// TIA Portal project "Elevator" (V15)

(* hardware
DEVICE "S7-1200 station_1"  S7-1200 Station
   slot 0: "Rack_0"  S7-1200 Rack  Rack  V1.0
   slot 1: "PLC_1"  CPU 1215C DC/DC/Rly  6ES7 215-1HG40-0XB0  V4.2
DEVICE "HMI_1"  KTP700 Basic PN
   slot 0: "HMI_1"  KTP700 Basic PN  6AV2 123-2GB03-0AX0  15.0.0.0
   slot 1: "HMI_RT_1"  KTP700 Basic PN  6AV2 123-2GB03-0AX0  15.0.0.0
   slot 5: "HMI_1.IE_CP_1"  PROFINET Interface  15.0.0.0
      slot 1: "PROFINET Interface_1"  PROFINET Interface
         slot 1: "Port_1"  Port
*)

// ===== PLC "PLC_1"  CPU 1215C DC/DC/Rly =====

VAR_GLOBAL   // PLC tag table "Default tag table"
   "asansor_tus_F1" AT %I4.0 : Bool;
   "kat_cagri_F1" AT %I4.5 : Bool;
   "kat_1" AT %M0.0 : Bool;
   "asansor_tus_F2" AT %I4.1 : Bool;
   "kat_cagri_F2" AT %I4.6 : Bool;
   "kat_2" AT %M0.1 : Bool;
   "asansor_tus_F3" AT %I4.2 : Bool;
   "kat_cagri_F3" AT %I4.7 : Bool;
   "kat_3" AT %M0.2 : Bool;
   "asansor_tus_F4" AT %I4.3 : Bool;
   "kat_cagri_F4" AT %I5.0 : Bool;
   "kat_4" AT %M0.3 : Bool;
   "Clock_1Hz" AT %M100.5 : Bool;
   "Motor_Yukari" AT %Q7.1 : Bool;
   "Motor_Asagi" AT %Q7.2 : Bool;
   "bas_sayaci" AT %MW10 : UInt;
   "System_Byte" AT %MB100 : Byte;
   "FirstScan" AT %M100.0 : Bool;
   "DiagStatusUpdate" AT %M100.1 : Bool;
   "AlwaysTRUE" AT %M100.2 : Bool;
   "AlwaysFALSE" AT %M100.3 : Bool;
   "Clock_Byte" AT %MB100 : Byte;
   "Clock_10Hz" AT %M100.0 : Bool;
   "Clock_5Hz" AT %M100.1 : Bool;
   "Clock_2.5Hz" AT %M100.2 : Bool;
   "Clock_2Hz" AT %M100.3 : Bool;
   "Clock_1.25Hz" AT %M100.4 : Bool;
   "Clock_0.625Hz" AT %M100.6 : Bool;
   "Clock_0.5Hz" AT %M100.7 : Bool;
   "F1_sensor" AT %I6.0 : Bool;
   "F2_sensor" AT %I6.1 : Bool;
   "F4_sensor" AT %I6.3 : Bool;
   "F3_sensor" AT %I6.2 : Bool;
   "F5_sensor" AT %I6.4 : Bool;
   "yon_yukari" AT %M0.5 : Bool;
   "yon_asagi" AT %M0.6 : Bool;
   "kat_5" AT %M0.4 : Bool;
   "asansor_tus_F5" AT %I4.4 : Bool;
   "kat_cagri_F5" AT %I5.1 : Bool;
   "kapi_kapaniyor" AT %M2.1 : Bool;
   "kapi_motoru" AT %Q7.0 : Bool;
   "kapi_acik_F3" AT %M1.2 : Bool;
   "kapi_kapandi" AT %M2.0 : Bool;
   "kapi_acik_F4" AT %M1.3 : Bool;
   "kapi_acik_F2" AT %M1.1 : Bool;
   "kapi_acik_F1" AT %M1.0 : Bool;
   "kapi_acik_F5" AT %M1.4 : Bool;
   "acma_tusu" AT %I5.2 : Bool;
   "engel_sensor" AT %I5.4 : Bool;
   "agirlik_sensor" AT %I5.5 : Bool;
   "kapi_tekrar_acildi" AT %M2.3 : Bool;
   "kapama_tusu" AT %I5.3 : Bool;
   "Tag_1" AT %M1.5 : Bool;
   "Tag_2" AT %M1.6 : Bool;
END_VAR

// folder: System blocks/Program resources

DATA_BLOCK "delay_reset5"   // DB1
{ S7_Optimized_Access := 'TRUE' }
AUTHOR : Simatic
FAMILY : IEC
NAME : IEC_TMR
VERSION : 1.0
// stored: InstanceOfName IEC_TIMER
"IEC_TIMER"
BEGIN
END_DATA_BLOCK

DATA_BLOCK "delay_reset4"   // DB2
{ S7_Optimized_Access := 'TRUE' }
AUTHOR : Simatic
FAMILY : IEC
NAME : IEC_TMR
VERSION : 1.0
// stored: InstanceOfName IEC_TIMER
"IEC_TIMER"
BEGIN
END_DATA_BLOCK

DATA_BLOCK "delay_reset3"   // DB3
{ S7_Optimized_Access := 'TRUE' }
AUTHOR : Simatic
FAMILY : IEC
NAME : IEC_TMR
VERSION : 1.0
// stored: InstanceOfName IEC_TIMER
"IEC_TIMER"
BEGIN
END_DATA_BLOCK

DATA_BLOCK "delay_reset2"   // DB4
{ S7_Optimized_Access := 'TRUE' }
AUTHOR : Simatic
FAMILY : IEC
NAME : IEC_TMR
VERSION : 1.0
// stored: InstanceOfName IEC_TIMER
"IEC_TIMER"
BEGIN
END_DATA_BLOCK

DATA_BLOCK "kapi_acik_zamani"   // DB5
{ S7_Optimized_Access := 'TRUE' }
AUTHOR : Simatic
FAMILY : IEC
NAME : IEC_TMR
VERSION : 1.0
// stored: InstanceOfName IEC_TIMER
"IEC_TIMER"
BEGIN
END_DATA_BLOCK

DATA_BLOCK "kapi_kapanma_zamani"   // DB6
{ S7_Optimized_Access := 'TRUE' }
AUTHOR : Simatic
FAMILY : IEC
NAME : IEC_TMR
VERSION : 1.0
// stored: InstanceOfName IEC_TIMER
"IEC_TIMER"
BEGIN
END_DATA_BLOCK

DATA_BLOCK "reset_acilma_zamani"   // DB7
{ S7_Optimized_Access := 'TRUE' }
AUTHOR : Simatic
FAMILY : IEC
NAME : IEC_TMR
VERSION : 1.0
// stored: InstanceOfName IEC_TIMER
"IEC_TIMER"
BEGIN
END_DATA_BLOCK

DATA_BLOCK "reset_kapama_tusu"   // DB8
{ S7_Optimized_Access := 'TRUE' }
AUTHOR : Simatic
FAMILY : IEC
NAME : IEC_TMR
VERSION : 1.0
// stored: InstanceOfName IEC_TIMER
"IEC_TIMER"
BEGIN
END_DATA_BLOCK

DATA_BLOCK "delay_reset1"   // DB9
{ S7_Optimized_Access := 'TRUE' }
AUTHOR : Simatic
FAMILY : IEC
NAME : IEC_TMR
VERSION : 1.0
// stored: InstanceOfName IEC_TIMER
"IEC_TIMER"
BEGIN
END_DATA_BLOCK

// folder: (top level)

ORGANIZATION_BLOCK "Main"   // OB1, LAD, ProgramCycle
TITLE = "Main Program Sweep (Cycle)"
{ S7_Optimized_Access := 'TRUE' }
VERSION : 0.1
   VAR_INPUT
      Initial_Call : Bool;   // Initial call of this OB
      Remanence : Bool;   // =True, if remanent data are available
   END_VAR
   VAR_TEMP   // added for the SCL form of the ladder/FBD networks
      _w1 : Bool;
      _w2 : Bool;
      _w3 : Bool;
      _w4 : Bool;
      _w5 : Bool;
   END_VAR
BEGIN

REGION Network 1: Asansör Çağrıları
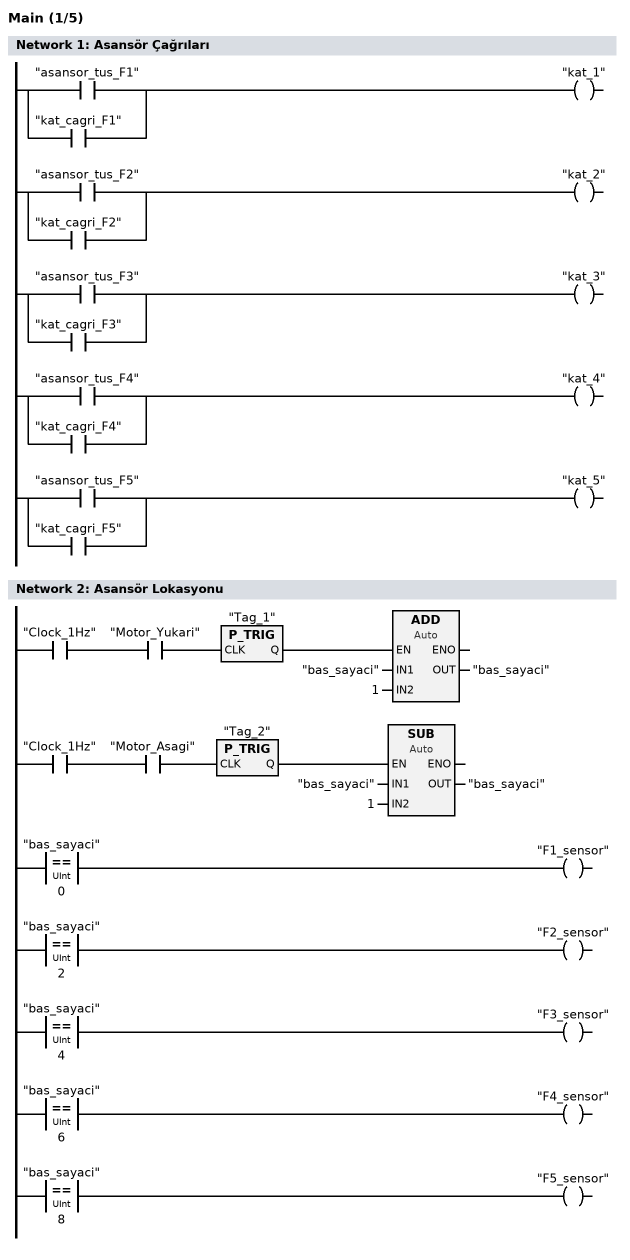
   RUNG wire#powerrail
      Contact( "asansor_tus_F1" )
      wire#w1
      Coil( "kat_1" )
   END_RUNG
   RUNG wire#powerrail
      Contact( "kat_cagri_F1" )
   END_RUNG wire#w1
   RUNG wire#powerrail
      Contact( "asansor_tus_F2" )
      wire#w2
      Coil( "kat_2" )
   END_RUNG
   RUNG wire#powerrail
      Contact( "kat_cagri_F2" )
   END_RUNG wire#w2
   RUNG wire#powerrail
      Contact( "asansor_tus_F3" )
      wire#w3
      Coil( "kat_3" )
   END_RUNG
   RUNG wire#powerrail
      Contact( "kat_cagri_F3" )
   END_RUNG wire#w3
   RUNG wire#powerrail
      Contact( "asansor_tus_F4" )
      wire#w4
      Coil( "kat_4" )
   END_RUNG
   RUNG wire#powerrail
      Contact( "kat_cagri_F4" )
   END_RUNG wire#w4
   RUNG wire#powerrail
      Contact( "asansor_tus_F5" )
      wire#w5
      Coil( "kat_5" )
   END_RUNG
   RUNG wire#powerrail
      Contact( "kat_cagri_F5" )
   END_RUNG wire#w5
   // the same network as SCL:
   "kat_1" := "asansor_tus_F1" OR "kat_cagri_F1";
   "kat_2" := "asansor_tus_F2" OR "kat_cagri_F2";
   "kat_3" := "asansor_tus_F3" OR "kat_cagri_F3";
   "kat_4" := "asansor_tus_F4" OR "kat_cagri_F4";
   "kat_5" := "asansor_tus_F5" OR "kat_cagri_F5";
END_REGION

REGION Network 2: Asansör Lokasyonu
   RUNG wire#powerrail
      Contact( "Clock_1Hz" )
      Contact( "Motor_Yukari" )
      P_Trig( "Tag_1" )
      Add(in1 := "bas_sayaci", in2 := 1, out => "bas_sayaci")
   END_RUNG
   RUNG wire#powerrail
      Contact( "Clock_1Hz" )
      Contact( "Motor_Asagi" )
      P_Trig( "Tag_2" )
      Sub(in1 := "bas_sayaci", in2 := 1, out => "bas_sayaci")
   END_RUNG
   RUNG wire#powerrail
      { S7_Templates := "SrcType := UInt" } EQ_Contact(in1 := "bas_sayaci", in2 := 0)
      Coil( "F1_sensor" )
   END_RUNG
   RUNG wire#powerrail
      { S7_Templates := "SrcType := UInt" } EQ_Contact(in1 := "bas_sayaci", in2 := 2)
      Coil( "F2_sensor" )
   END_RUNG
   RUNG wire#powerrail
      { S7_Templates := "SrcType := UInt" } EQ_Contact(in1 := "bas_sayaci", in2 := 4)
      Coil( "F3_sensor" )
   END_RUNG
   RUNG wire#powerrail
      { S7_Templates := "SrcType := UInt" } EQ_Contact(in1 := "bas_sayaci", in2 := 6)
      Coil( "F4_sensor" )
   END_RUNG
   RUNG wire#powerrail
      { S7_Templates := "SrcType := UInt" } EQ_Contact(in1 := "bas_sayaci", in2 := 8)
      Coil( "F5_sensor" )
   END_RUNG
   // the same network as SCL:
   #_w1 := "Clock_1Hz" AND "Motor_Yukari";
   #_w2 := #_w1 AND NOT "Tag_1";   // rising edge
   "Tag_1" := #_w1;
   IF #_w2 THEN "bas_sayaci" := "bas_sayaci" + 1; END_IF;
   #_w3 := "Clock_1Hz" AND "Motor_Asagi";
   #_w4 := #_w3 AND NOT "Tag_2";   // rising edge
   "Tag_2" := #_w3;
   IF #_w4 THEN "bas_sayaci" := "bas_sayaci" - 1; END_IF;
   "F1_sensor" := "bas_sayaci" = 0;
   "F2_sensor" := "bas_sayaci" = 2;
   "F3_sensor" := "bas_sayaci" = 4;
   "F4_sensor" := "bas_sayaci" = 6;
   "F5_sensor" := "bas_sayaci" = 8;
END_REGION

REGION Network 3: Asansör Yönelimi
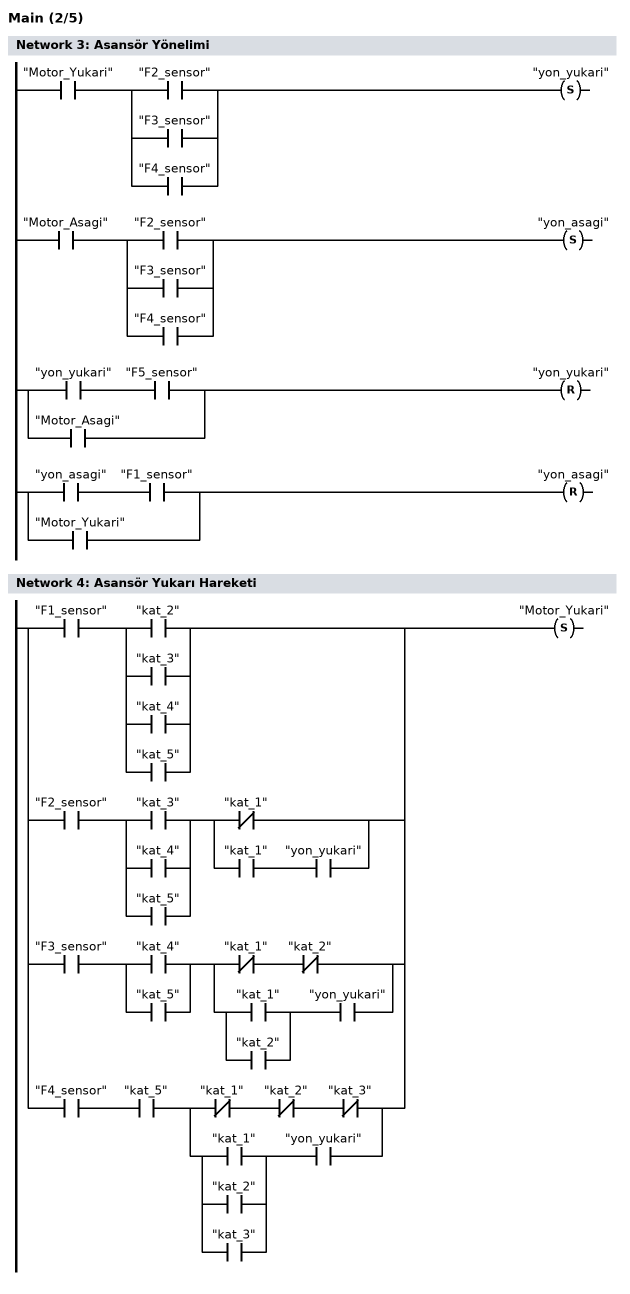
   RUNG wire#powerrail
      Contact( "Motor_Yukari" )
      wire#w1
      Contact( "F2_sensor" )
      wire#w2
      S_Coil( "yon_yukari" )
   END_RUNG
   RUNG wire#w1
      Contact( "F3_sensor" )
   END_RUNG wire#w2
   RUNG wire#w1
      Contact( "F4_sensor" )
   END_RUNG wire#w2
   RUNG wire#powerrail
      Contact( "Motor_Asagi" )
      wire#w3
      Contact( "F2_sensor" )
      wire#w4
      S_Coil( "yon_asagi" )
   END_RUNG
   RUNG wire#w3
      Contact( "F3_sensor" )
   END_RUNG wire#w4
   RUNG wire#w3
      Contact( "F4_sensor" )
   END_RUNG wire#w4
   RUNG wire#powerrail
      Contact( "yon_yukari" )
      Contact( "F5_sensor" )
      wire#w5
      R_Coil( "yon_yukari" )
   END_RUNG
   RUNG wire#powerrail
      Contact( "Motor_Asagi" )
   END_RUNG wire#w5
   RUNG wire#powerrail
      Contact( "yon_asagi" )
      Contact( "F1_sensor" )
      wire#w6
      R_Coil( "yon_asagi" )
   END_RUNG
   RUNG wire#powerrail
      Contact( "Motor_Yukari" )
   END_RUNG wire#w6
   // the same network as SCL:
   IF "Motor_Yukari" AND ("F2_sensor" OR "F3_sensor" OR "F4_sensor") THEN "yon_yukari" := TRUE; END_IF;
   IF "Motor_Asagi" AND ("F2_sensor" OR "F3_sensor" OR "F4_sensor") THEN "yon_asagi" := TRUE; END_IF;
   IF ("yon_yukari" AND "F5_sensor") OR "Motor_Asagi" THEN "yon_yukari" := FALSE; END_IF;
   IF ("yon_asagi" AND "F1_sensor") OR "Motor_Yukari" THEN "yon_asagi" := FALSE; END_IF;
END_REGION

REGION Network 4: Asansör Yukarı Hareketi
   RUNG wire#powerrail
      Contact( "F1_sensor" )
      wire#w1
      Contact( "kat_2" )
      wire#w2
      S_Coil( "Motor_Yukari" )
   END_RUNG
   RUNG wire#w1
      Contact( "kat_3" )
   END_RUNG wire#w2
   RUNG wire#w1
      Contact( "kat_4" )
   END_RUNG wire#w2
   RUNG wire#w1
      Contact( "kat_5" )
   END_RUNG wire#w2
   RUNG wire#powerrail
      Contact( "F2_sensor" )
      wire#w3
      Contact( "kat_3" )
      wire#w4
      I_Contact( "kat_1" )
   END_RUNG wire#w2
   RUNG wire#w3
      Contact( "kat_4" )
   END_RUNG wire#w4
   RUNG wire#w3
      Contact( "kat_5" )
   END_RUNG wire#w4
   RUNG wire#w4
      Contact( "kat_1" )
      Contact( "yon_yukari" )
   END_RUNG wire#w2
   RUNG wire#powerrail
      Contact( "F3_sensor" )
      wire#w5
      Contact( "kat_4" )
      wire#w6
      I_Contact( "kat_1" )
      I_Contact( "kat_2" )
   END_RUNG wire#w2
   RUNG wire#w5
      Contact( "kat_5" )
   END_RUNG wire#w6
   RUNG wire#w6
      Contact( "kat_1" )
      wire#w7
      Contact( "yon_yukari" )
   END_RUNG wire#w2
   RUNG wire#w6
      Contact( "kat_2" )
   END_RUNG wire#w7
   RUNG wire#powerrail
      Contact( "F4_sensor" )
      Contact( "kat_5" )
      wire#w8
      I_Contact( "kat_1" )
      I_Contact( "kat_2" )
      I_Contact( "kat_3" )
   END_RUNG wire#w2
   RUNG wire#w8
      Contact( "kat_1" )
      wire#w9
      Contact( "yon_yukari" )
   END_RUNG wire#w2
   RUNG wire#w8
      Contact( "kat_2" )
   END_RUNG wire#w9
   RUNG wire#w8
      Contact( "kat_3" )
   END_RUNG wire#w9
   // the same network as SCL:
   IF ("F1_sensor" AND ("kat_2" OR "kat_3" OR "kat_4" OR "kat_5")) OR ("F2_sensor" AND ("kat_3" OR "kat_4" OR "kat_5") AND (NOT "kat_1" OR ("kat_1" AND "yon_yukari"))) OR ("F3_sensor" AND ("kat_4" OR "kat_5") AND ((NOT "kat_1" AND NOT "kat_2") OR (("kat_1" OR "kat_2") AND "yon_yukari"))) OR ("F4_sensor" AND "kat_5" AND ((NOT "kat_1" AND NOT "kat_2" AND NOT "kat_3") OR (("kat_1" OR "kat_2" OR "kat_3") AND "yon_yukari"))) THEN
       "Motor_Yukari" := TRUE;
   END_IF;
END_REGION

REGION Network 5: Asansör Aşağı Hareketi
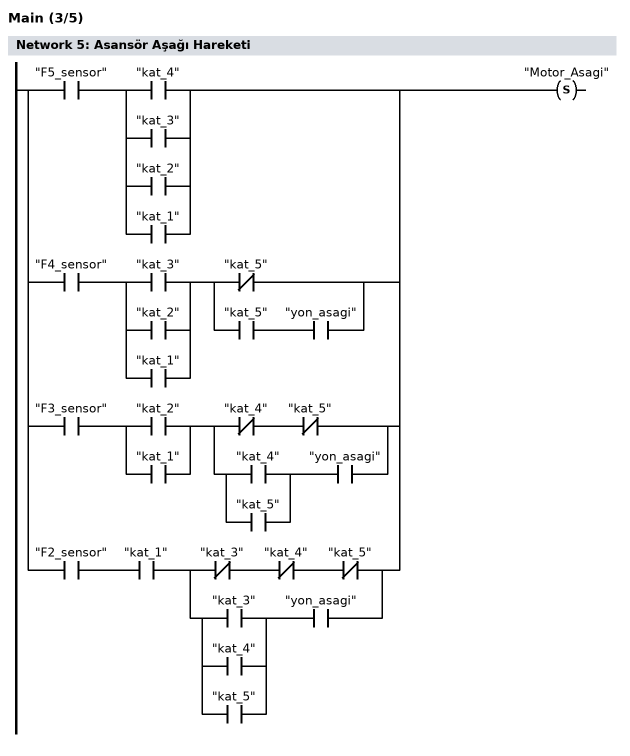
   RUNG wire#powerrail
      Contact( "F5_sensor" )
      wire#w1
      Contact( "kat_4" )
      wire#w2
      S_Coil( "Motor_Asagi" )
   END_RUNG
   RUNG wire#w1
      Contact( "kat_3" )
   END_RUNG wire#w2
   RUNG wire#w1
      Contact( "kat_2" )
   END_RUNG wire#w2
   RUNG wire#w1
      Contact( "kat_1" )
   END_RUNG wire#w2
   RUNG wire#powerrail
      Contact( "F4_sensor" )
      wire#w3
      Contact( "kat_3" )
      wire#w4
      I_Contact( "kat_5" )
   END_RUNG wire#w2
   RUNG wire#w3
      Contact( "kat_2" )
   END_RUNG wire#w4
   RUNG wire#w3
      Contact( "kat_1" )
   END_RUNG wire#w4
   RUNG wire#w4
      Contact( "kat_5" )
      Contact( "yon_asagi" )
   END_RUNG wire#w2
   RUNG wire#powerrail
      Contact( "F3_sensor" )
      wire#w5
      Contact( "kat_2" )
      wire#w6
      I_Contact( "kat_4" )
      I_Contact( "kat_5" )
   END_RUNG wire#w2
   RUNG wire#w5
      Contact( "kat_1" )
   END_RUNG wire#w6
   RUNG wire#w6
      Contact( "kat_4" )
      wire#w7
      Contact( "yon_asagi" )
   END_RUNG wire#w2
   RUNG wire#w6
      Contact( "kat_5" )
   END_RUNG wire#w7
   RUNG wire#powerrail
      Contact( "F2_sensor" )
      Contact( "kat_1" )
      wire#w8
      I_Contact( "kat_3" )
      I_Contact( "kat_4" )
      I_Contact( "kat_5" )
   END_RUNG wire#w2
   RUNG wire#w8
      Contact( "kat_3" )
      wire#w9
      Contact( "yon_asagi" )
   END_RUNG wire#w2
   RUNG wire#w8
      Contact( "kat_4" )
   END_RUNG wire#w9
   RUNG wire#w8
      Contact( "kat_5" )
   END_RUNG wire#w9
   // the same network as SCL:
   IF ("F5_sensor" AND ("kat_4" OR "kat_3" OR "kat_2" OR "kat_1")) OR ("F4_sensor" AND ("kat_3" OR "kat_2" OR "kat_1") AND (NOT "kat_5" OR ("kat_5" AND "yon_asagi"))) OR ("F3_sensor" AND ("kat_2" OR "kat_1") AND ((NOT "kat_4" AND NOT "kat_5") OR (("kat_4" OR "kat_5") AND "yon_asagi"))) OR ("F2_sensor" AND "kat_1" AND ((NOT "kat_3" AND NOT "kat_4" AND NOT "kat_5") OR (("kat_3" OR "kat_4" OR "kat_5") AND "yon_asagi"))) THEN
       "Motor_Asagi" := TRUE;
   END_IF;
END_REGION

REGION Network 6: Asansör Durma - Kapı Açılması
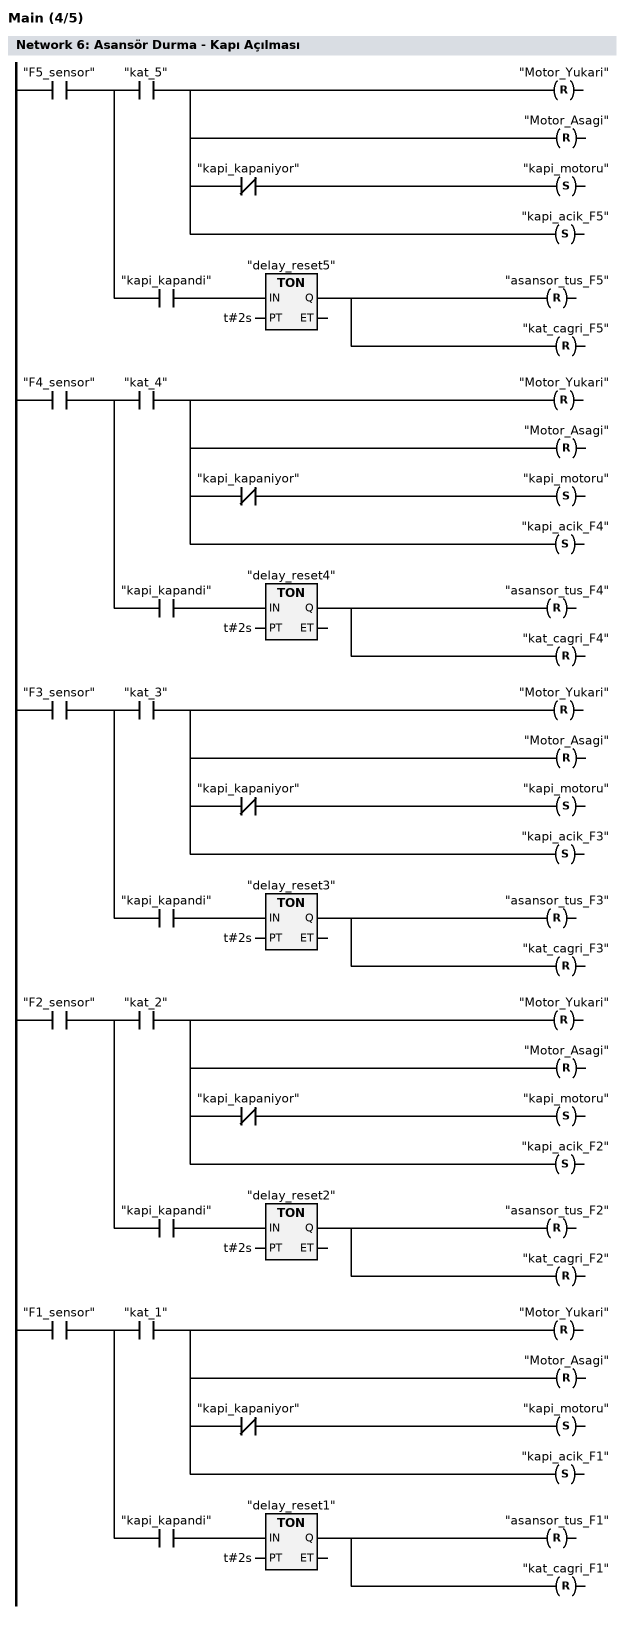
   #_w1 := "F5_sensor" AND "kat_5";
   IF #_w1 THEN
       "Motor_Yukari" := FALSE;
       "Motor_Asagi" := FALSE;
   END_IF;
   IF #_w1 AND NOT "kapi_kapaniyor" THEN "kapi_motoru" := TRUE; END_IF;
   IF #_w1 THEN "kapi_acik_F5" := TRUE; END_IF;
   "delay_reset5".TON(IN := "F5_sensor" AND "kapi_kapandi", PT := t#2s);
   IF "delay_reset5".Q THEN
       "asansor_tus_F5" := FALSE;
       "kat_cagri_F5" := FALSE;
   END_IF;
   #_w2 := "F4_sensor" AND "kat_4";
   IF #_w2 THEN
       "Motor_Yukari" := FALSE;
       "Motor_Asagi" := FALSE;
   END_IF;
   IF #_w2 AND NOT "kapi_kapaniyor" THEN "kapi_motoru" := TRUE; END_IF;
   IF #_w2 THEN "kapi_acik_F4" := TRUE; END_IF;
   "delay_reset4".TON(IN := "F4_sensor" AND "kapi_kapandi", PT := t#2s);
   IF "delay_reset4".Q THEN
       "asansor_tus_F4" := FALSE;
       "kat_cagri_F4" := FALSE;
   END_IF;
   #_w3 := "F3_sensor" AND "kat_3";
   IF #_w3 THEN
       "Motor_Yukari" := FALSE;
       "Motor_Asagi" := FALSE;
   END_IF;
   IF #_w3 AND NOT "kapi_kapaniyor" THEN "kapi_motoru" := TRUE; END_IF;
   IF #_w3 THEN "kapi_acik_F3" := TRUE; END_IF;
   "delay_reset3".TON(IN := "F3_sensor" AND "kapi_kapandi", PT := t#2s);
   IF "delay_reset3".Q THEN
       "asansor_tus_F3" := FALSE;
       "kat_cagri_F3" := FALSE;
   END_IF;
   #_w4 := "F2_sensor" AND "kat_2";
   IF #_w4 THEN
       "Motor_Yukari" := FALSE;
       "Motor_Asagi" := FALSE;
   END_IF;
   IF #_w4 AND NOT "kapi_kapaniyor" THEN "kapi_motoru" := TRUE; END_IF;
   IF #_w4 THEN "kapi_acik_F2" := TRUE; END_IF;
   "delay_reset2".TON(IN := "F2_sensor" AND "kapi_kapandi", PT := t#2s);
   IF "delay_reset2".Q THEN
       "asansor_tus_F2" := FALSE;
       "kat_cagri_F2" := FALSE;
   END_IF;
   #_w5 := "F1_sensor" AND "kat_1";
   IF #_w5 THEN
       "Motor_Yukari" := FALSE;
       "Motor_Asagi" := FALSE;
   END_IF;
   IF #_w5 AND NOT "kapi_kapaniyor" THEN "kapi_motoru" := TRUE; END_IF;
   IF #_w5 THEN "kapi_acik_F1" := TRUE; END_IF;
   "delay_reset1".TON(IN := "F1_sensor" AND "kapi_kapandi", PT := t#2s);
   IF "delay_reset1".Q THEN
       "asansor_tus_F1" := FALSE;
       "kat_cagri_F1" := FALSE;
   END_IF;
END_REGION

REGION Network 7: Asansör Kapı Kapanması
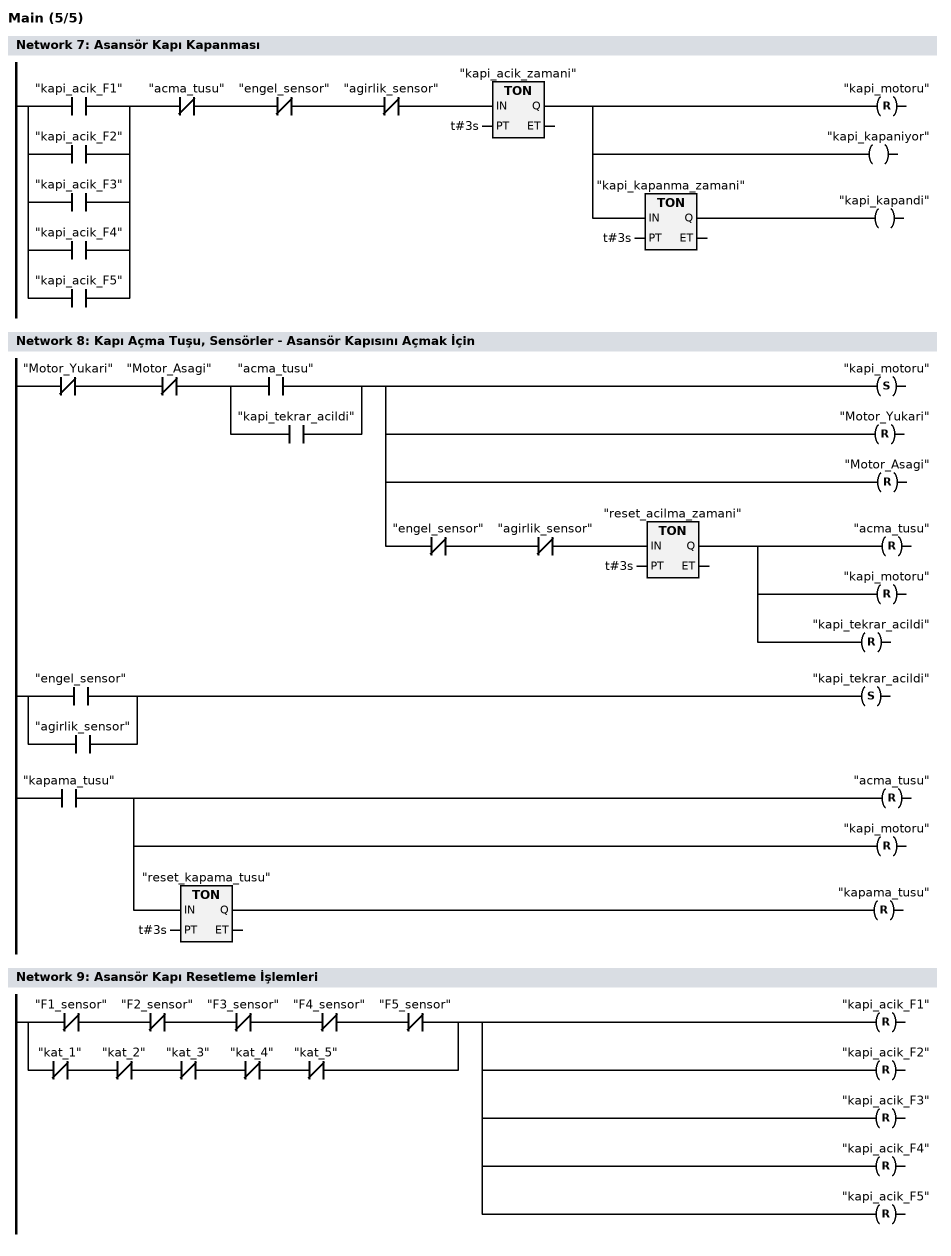
   "kapi_acik_zamani".TON(IN := ("kapi_acik_F1" OR "kapi_acik_F2" OR "kapi_acik_F3" OR "kapi_acik_F4" OR "kapi_acik_F5") AND NOT "acma_tusu" AND NOT "engel_sensor" AND NOT "agirlik_sensor",
                          PT := t#3s);
   IF "kapi_acik_zamani".Q THEN "kapi_motoru" := FALSE; END_IF;
   "kapi_kapaniyor" := "kapi_acik_zamani".Q;
   "kapi_kapanma_zamani".TON(IN := "kapi_acik_zamani".Q, PT := t#3s);
   "kapi_kapandi" := "kapi_kapanma_zamani".Q;
END_REGION

REGION Network 8: Kapı Açma Tuşu, Sensörler - Asansör Kapısını Açmak İçin
   #_w1 := NOT "Motor_Yukari" AND NOT "Motor_Asagi" AND ("acma_tusu" OR "kapi_tekrar_acildi");
   IF #_w1 THEN
       "kapi_motoru" := TRUE;
       "Motor_Yukari" := FALSE;
       "Motor_Asagi" := FALSE;
   END_IF;
   "reset_acilma_zamani".TON(IN := #_w1 AND NOT "engel_sensor" AND NOT "agirlik_sensor", PT := t#3s);
   IF "reset_acilma_zamani".Q THEN
       "acma_tusu" := FALSE;
       "kapi_motoru" := FALSE;
       "kapi_tekrar_acildi" := FALSE;
   END_IF;
   IF "engel_sensor" OR "agirlik_sensor" THEN "kapi_tekrar_acildi" := TRUE; END_IF;
   IF "kapama_tusu" THEN
       "acma_tusu" := FALSE;
       "kapi_motoru" := FALSE;
   END_IF;
   "reset_kapama_tusu".TON(IN := "kapama_tusu", PT := t#3s);
   IF "reset_kapama_tusu".Q THEN "kapama_tusu" := FALSE; END_IF;
END_REGION

REGION Network 9: Asansör Kapı Resetleme İşlemleri
   RUNG wire#powerrail
      I_Contact( "F1_sensor" )
      I_Contact( "F2_sensor" )
      I_Contact( "F3_sensor" )
      I_Contact( "F4_sensor" )
      I_Contact( "F5_sensor" )
      wire#w1
      R_Coil( "kapi_acik_F1" )
   END_RUNG
   RUNG wire#powerrail
      I_Contact( "kat_1" )
      I_Contact( "kat_2" )
      I_Contact( "kat_3" )
      I_Contact( "kat_4" )
      I_Contact( "kat_5" )
   END_RUNG wire#w1
   RUNG wire#w1
      R_Coil( "kapi_acik_F2" )
   END_RUNG
   RUNG wire#w1
      R_Coil( "kapi_acik_F3" )
   END_RUNG
   RUNG wire#w1
      R_Coil( "kapi_acik_F4" )
   END_RUNG
   RUNG wire#w1
      R_Coil( "kapi_acik_F5" )
   END_RUNG
   // the same network as SCL:
   IF (NOT "F1_sensor" AND NOT "F2_sensor" AND NOT "F3_sensor" AND NOT "F4_sensor" AND NOT "F5_sensor") OR (NOT "kat_1" AND NOT "kat_2" AND NOT "kat_3" AND NOT "kat_4" AND NOT "kat_5") THEN
       "kapi_acik_F1" := FALSE;
       "kapi_acik_F2" := FALSE;
       "kapi_acik_F3" := FALSE;
       "kapi_acik_F4" := FALSE;
       "kapi_acik_F5" := FALSE;
   END_IF;
END_REGION
END_ORGANIZATION_BLOCK

(* ===== HMI "HMI_RT_1" =====
system functions are stored by id; their names below are inferred from use
connection "HMI_Connection_1": ETHERNET, SMART_S7_1200_OMS

HMI tags "Default tag table"
   "Tag_ScreenNumber" : UInt, internal
   "kat_1" : Bool = PLC kat_1 AT %M0.0, 1 s
   "kat_2" : Bool = PLC kat_2 AT %M0.1, 1 s
   "kat_3" : Bool = PLC kat_3 AT %M0.2, 1 s
   "kat_4" : Bool = PLC kat_4 AT %M0.3, 1 s
   "kat_5" : Bool = PLC kat_5 AT %M0.4, 1 s
   "engel_sensor" : Bool = PLC engel_sensor AT %I5.4, 1 s
   "agirlik_sensor" : Bool = PLC agirlik_sensor AT %I5.5, 1 s
   "F5_sensor" : Bool = PLC F5_sensor AT %I6.4, 1 s
   "F4_sensor" : Bool = PLC F4_sensor AT %I6.3, 1 s
   "F3_sensor" : Bool = PLC F3_sensor AT %I6.2, 1 s
   "F2_sensor" : Bool = PLC F2_sensor AT %I6.1, 1 s
   "F1_sensor" : Bool = PLC F1_sensor AT %I6.0, 1 s
   "Motor_Yukari" : Bool = PLC Motor_Yukari AT %Q7.1, 1 s
   "Motor_Asagi" : Bool = PLC Motor_Asagi AT %Q7.2, 1 s
   "kapi_kapaniyor" : Bool = PLC kapi_kapaniyor AT %M2.1, 1 s
   "kapi_motoru" : Bool = PLC kapi_motoru AT %Q7.0, 1 s
   "kat_cagri_F5" : Bool = PLC kat_cagri_F5 AT %I5.1, 1 s
   "kat_cagri_F4" : Bool = PLC kat_cagri_F4 AT %I5.0, 1 s
   "kat_cagri_F3" : Bool = PLC kat_cagri_F3 AT %I4.7, 1 s
   "kat_cagri_F2" : Bool = PLC kat_cagri_F2 AT %I4.6, 1 s
   "kat_cagri_F1" : Bool = PLC kat_cagri_F1 AT %I4.5, 1 s
   "asansor_tus_F1" : Bool = PLC asansor_tus_F1 AT %I4.0, 1 s
   "asansor_tus_F2" : Bool = PLC asansor_tus_F2 AT %I4.1, 1 s
   "asansor_tus_F3" : Bool = PLC asansor_tus_F3 AT %I4.2, 1 s
   "asansor_tus_F4" : Bool = PLC asansor_tus_F4 AT %I4.3, 1 s
   "asansor_tus_F5" : Bool = PLC asansor_tus_F5 AT %I4.4, 1 s
   "acma_tusu" : Bool = PLC acma_tusu AT %I5.2, 1 s
   "kapama_tusu" : Bool = PLC kapama_tusu AT %I5.3, 1 s

Template "Template_1" 800x480
   Button "Exit" at 714,429 size 71x50; TextOff 'Exit'; PictureOff "ExitRuntime_KTP700_Basic_PN_TR"; PictureOn "ExitRuntime_KTP700_Basic_PN_TR"
      on Release: StopRuntime(0)
   Button "Template_Button" at 614,429 size 71x50; TextOff 'Text'
   Button "Template_Button_1" at 514,429 size 71x50; TextOff 'Text'
   Button "Template_Button_2" at 414,429 size 71x50; TextOff 'Text'
   Button "Template_Button_3" at 314,429 size 71x50; TextOff 'Text'
   Button "Template_Button_4" at 214,429 size 71x50; TextOff 'Text'
   Button "Alarms" at 114,429 size 71x50; TextOff 'Alarms'; PictureOff "AlarmDisplay_KTP700_Basic_PN_TR"; PictureOn "AlarmDisplay_KTP700_Basic_PN_TR"
      on Release: function_ef3f5d25("Alarm window_Unacknowledged", -1)
   Button "Start screen" at 14,429 size 71x50; TextOff 'Start screen'; PictureOff "NavigateHome_KTP700_Basic_PN_TR"; PictureOn "NavigateHome_KTP700_Basic_PN_TR"
      on Release: ActivateScreen("Root screen", 0)
   SymbolicIOField "Symbolic_IO_Field_Screen" at 93,9 size 600x33; TextOff '0'; TextOn '1'; TextList "TextList_ScreenNames"
      ProcessValue <- "Tag_ScreenNumber"
      on Change: ActivateScreenByNumber("Tag_ScreenNumber", 0)
   DateTimeField "HmiScreenItemData" at 695,25 size 105x25
   DateTimeField "HmiScreenItemData_1" at 695,0 size 105x25
   GraphicView "Logo" at 0,0 size 91x51; Picture "Logo of HMI_1"

screen "Root screen" 800x480, template "Template_1"
   on GenerateScreen: SetTag("Tag_ScreenNumber", 1)
   Button "Button_1" at 623,54 size 146x32; TextOff 'Asansör Konumu'
   Button "Button_2" at 16,54 size 152x32; TextOn 'Kat Tuşları'; TextOff 'Kat Tuşları'
   Button "Button_3" at 190,54 size 152x32; TextOn 'Asansördeki Tuşlar'; TextOff 'Asansördeki Tuşlar'
   Button "Button_4" at 364,54 size 152x32; TextOn 'Sensörler'; TextOff 'Sensörler'
   Button "Button_5" at 623,94 size 145x24; TextOff 'Kat 5'
      Appearance <- "F5_sensor"
   Button "Button_10" at 16,91 size 152x28; TextOn '5. Kat Tuşu'; TextOff '5. Kat Tuşu'
      Appearance <- "kat_5"
      on Press: SetBit("kat_cagri_F5")
   Button "Button_15" at 189,91 size 40x28; TextOn '5'; TextOff '5'
      on Press: SetBit("asansor_tus_F5")
      Appearance <- "kat_5"
   Button "Button_20" at 249,91 size 93x32; TextOn 'Kapı Aç'; TextOff 'Kapı Aç'
      on Press: SetBit("acma_tusu")
   Button "Button_21" at 249,129 size 93x32; TextOn 'Kapı Kapa'; TextOff 'Kapı Kapa'
      on Press: SetBit("kapama_tusu")
   Button "Button_22" at 624,251 size 147x32; TextOn 'Asansör Hareketi'; TextOff 'Asansör Hareketi'
   Button "Button_23" at 623,289 size 145x24; TextOn 'Yukarı Yönde'; TextOff 'Yukarı Yönde'
      Appearance <- "Motor_Yukari"
   Button "Button_6" at 623,125 size 145x24; TextOn 'Kat 4'; TextOff 'Kat 4'
      Appearance <- "F4_sensor"
   Button "Button_7" at 623,156 size 145x24; TextOn 'Kat 3'; TextOff 'Kat 3'
      Appearance <- "F3_sensor"
   Button "Button_8" at 623,187 size 145x24; TextOn 'Kat 2'; TextOff 'Kat 2'
      Appearance <- "F2_sensor"
   Button "Button_9" at 623,217 size 145x24; TextOn 'Kat 1'; TextOff 'Kat 1'
      Appearance <- "F1_sensor"
   Button "Button_11" at 624,323 size 145x24; TextOn 'Aşağı Yönde'; TextOff 'Aşağı Yönde'
      Appearance <- "Motor_Asagi"
   Button "Button_12" at 16,128 size 152x28; TextOn '4. Kat Tuşu'; TextOff '4. Kat Tuşu'
      Appearance <- "kat_4"
      on Press: SetBit("kat_cagri_F4")
   Button "Button_13" at 16,165 size 152x28; TextOn '3. Kat Tuşu'; TextOff '3. Kat Tuşu'
      Appearance <- "kat_3"
      on Press: SetBit("kat_cagri_F3")
   Button "Button_14" at 16,202 size 152x28; TextOn '2. Kat Tuşu'; TextOff '2. Kat Tuşu'
      Appearance <- "kat_2"
      on Press: SetBit("kat_cagri_F2")
   Button "Button_24" at 16,239 size 152x28; TextOn '1. Kat Tuşu'; TextOff '1. Kat Tuşu'
      Appearance <- "kat_1"
      on Press: SetBit("kat_cagri_F1")
   Button "Button_16" at 189,128 size 40x28; TextOn '4'; TextOff '4'
      on Press: SetBit("asansor_tus_F4")
      Appearance <- "kat_4"
   Button "Button_17" at 189,165 size 40x28; TextOn '3'; TextOff '3'
      Appearance <- "kat_3"
      on Press: SetBit("asansor_tus_F3")
   Button "Button_18" at 189,202 size 40x28; TextOn '2'; TextOff '2'
      on Press: SetBit("asansor_tus_F2")
      Appearance <- "kat_2"
   Button "Button_19" at 189,239 size 40x28; TextOn '1'; TextOff '1'
      Appearance <- "kat_1"
      on Press: SetBit("asansor_tus_F1")
   Button "Button_25" at 364,91 size 152x28; TextOn 'Engel Sensörü Aç'; TextOff 'Engel Sensörü Aç'
      on Press: SetTag("engel_sensor", 1)
      Appearance <- "engel_sensor"
   Button "Button_26" at 363,128 size 152x28; TextOn 'Engel Sensörü Kapa'; TextOff 'Engel Sensörü Kapa'
      on Press: SetTag("engel_sensor", 0)
      Appearance <- "engel_sensor"
   Button "Button_27" at 363,165 size 152x28; TextOn 'Ağırlık Sensörü Aç'; TextOff 'Ağırlık Sensörü Aç'
      on Press: SetTag("agirlik_sensor", 1)
      Appearance <- "agirlik_sensor"
   Button "Button_28" at 363,202 size 152x28; TextOn 'Ağırlık Sensörü Kapa'; TextOff 'Ağırlık Sensörü Kapa'
      on Press: SetTag("agirlik_sensor", 0)
      Appearance <- "agirlik_sensor"
   Button "Button_29" at 623,356 size 147x32; TextOn 'Kapı Durumu'; TextOff 'Kapı Durumu'
   Button "Button_30" at 624,394 size 70x24; TextOn 'Kapanıyor'; TextOff 'Kapanıyor'
      Appearance <- "kapi_kapaniyor"
   Button "Button_31" at 698,394 size 70x24; TextOn 'Açılıyor'; TextOff 'Açılıyor'
      Appearance <- "kapi_motoru"
*)